// TIA Portal V19 export
FUNCTION "FC70_RecordData" : Void   // FC70, LAD
{ S7_Optimized_Access := 'TRUE' }
// stored: AutoNumber false, SetENOAutomatically false
   VAR_TEMP   // added for the SCL form of the ladder/FBD networks
      _w1 : Bool;
   END_VAR
BEGIN

REGION Network 1: Record Production data
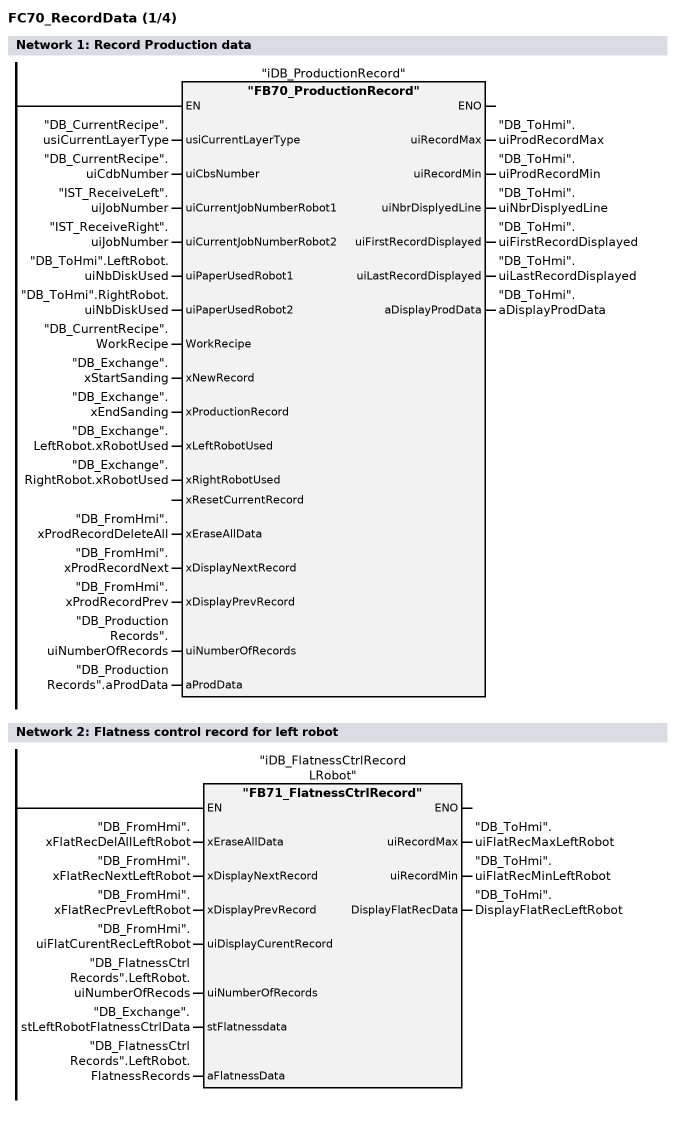
   RUNG wire#powerrail
      "iDB_ProductionRecord"(usiCurrentLayerType := "DB_CurrentRecipe".usiCurrentLayerType, uiCbsNumber := "DB_CurrentRecipe".uiCdbNumber, uiCurrentJobNumberRobot1 := "IST_ReceiveLeft".uiJobNumber, uiCurrentJobNumberRobot2 := "IST_ReceiveRight".uiJobNumber, uiPaperUsedRobot1 := "DB_ToHmi".LeftRobot.uiNbDiskUsed, uiPaperUsedRobot2 := "DB_ToHmi".RightRobot.uiNbDiskUsed, WorkRecipe := "DB_CurrentRecipe".WorkRecipe, xNewRecord := "DB_Exchange".xStartSanding, xProductionRecord := "DB_Exchange".xEndSanding, xLeftRobotUsed := "DB_Exchange".LeftRobot.xRobotUsed, xRightRobotUsed := "DB_Exchange".RightRobot.xRobotUsed, xResetCurrentRecord :=, xEraseAllData := "DB_FromHmi".xProdRecordDeleteAll, xDisplayNextRecord := "DB_FromHmi".xProdRecordNext, xDisplayPrevRecord := "DB_FromHmi".xProdRecordPrev, uiNumberOfRecords := "DB_ProductionRecords".uiNumberOfRecords, aProdData := "DB_ProductionRecords".aProdData, uiRecordMax => "DB_ToHmi".uiProdRecordMax, uiRecordMin => "DB_ToHmi".uiProdRecordMin, uiNbrDisplyedLine => "DB_ToHmi".uiNbrDisplyedLine, uiFirstRecordDisplayed => "DB_ToHmi".uiFirstRecordDisplayed, uiLastRecordDisplayed => "DB_ToHmi".uiLastRecordDisplayed, aDisplayProdData => "DB_ToHmi".aDisplayProdData)
   END_RUNG
   // the same network as SCL:
   "iDB_ProductionRecord"(usiCurrentLayerType := "DB_CurrentRecipe".usiCurrentLayerType,   // "FB70_ProductionRecord"
                          uiCbsNumber := "DB_CurrentRecipe".uiCdbNumber,
                          uiCurrentJobNumberRobot1 := "IST_ReceiveLeft".uiJobNumber,
                          uiCurrentJobNumberRobot2 := "IST_ReceiveRight".uiJobNumber,
                          uiPaperUsedRobot1 := "DB_ToHmi".LeftRobot.uiNbDiskUsed,
                          uiPaperUsedRobot2 := "DB_ToHmi".RightRobot.uiNbDiskUsed,
                          WorkRecipe := "DB_CurrentRecipe".WorkRecipe,
                          xNewRecord := "DB_Exchange".xStartSanding,
                          xProductionRecord := "DB_Exchange".xEndSanding,
                          xLeftRobotUsed := "DB_Exchange".LeftRobot.xRobotUsed,
                          xRightRobotUsed := "DB_Exchange".RightRobot.xRobotUsed,
                          xEraseAllData := "DB_FromHmi".xProdRecordDeleteAll,
                          xDisplayNextRecord := "DB_FromHmi".xProdRecordNext,
                          xDisplayPrevRecord := "DB_FromHmi".xProdRecordPrev,
                          uiNumberOfRecords := "DB_ProductionRecords".uiNumberOfRecords,
                          aProdData := "DB_ProductionRecords".aProdData,
                          uiRecordMax => "DB_ToHmi".uiProdRecordMax,
                          uiRecordMin => "DB_ToHmi".uiProdRecordMin,
                          uiNbrDisplyedLine => "DB_ToHmi".uiNbrDisplyedLine,
                          uiFirstRecordDisplayed => "DB_ToHmi".uiFirstRecordDisplayed,
                          uiLastRecordDisplayed => "DB_ToHmi".uiLastRecordDisplayed,
                          aDisplayProdData => "DB_ToHmi".aDisplayProdData);
END_REGION

REGION Network 2: Flatness control record for left robot
   RUNG wire#powerrail
      "iDB_FlatnessCtrlRecordLRobot"(xEraseAllData := "DB_FromHmi".xFlatRecDelAllLeftRobot, xDisplayNextRecord := "DB_FromHmi".xFlatRecNextLeftRobot, xDisplayPrevRecord := "DB_FromHmi".xFlatRecPrevLeftRobot, uiDisplayCurentRecord := "DB_FromHmi".uiFlatCurentRecLeftRobot, uiNumberOfRecords := "DB_FlatnessCtrlRecords".LeftRobot.uiNumberOfRecods, stFlatnessdata := "DB_Exchange".stLeftRobotFlatnessCtrlData, aFlatnessData := "DB_FlatnessCtrlRecords".LeftRobot.FlatnessRecords, uiRecordMax => "DB_ToHmi".uiFlatRecMaxLeftRobot, uiRecordMin => "DB_ToHmi".uiFlatRecMinLeftRobot, DisplayFlatRecData => "DB_ToHmi".DisplayFlatRecLeftRobot)
   END_RUNG
   // the same network as SCL:
   "iDB_FlatnessCtrlRecordLRobot"(xEraseAllData := "DB_FromHmi".xFlatRecDelAllLeftRobot,   // "FB71_FlatnessCtrlRecord"
                           xDisplayNextRecord := "DB_FromHmi".xFlatRecNextLeftRobot,
                           xDisplayPrevRecord := "DB_FromHmi".xFlatRecPrevLeftRobot,
                           uiDisplayCurentRecord := "DB_FromHmi".uiFlatCurentRecLeftRobot,
                           uiNumberOfRecords := "DB_FlatnessCtrlRecords".LeftRobot.uiNumberOfRecods,
                           stFlatnessdata := "DB_Exchange".stLeftRobotFlatnessCtrlData,
                           aFlatnessData := "DB_FlatnessCtrlRecords".LeftRobot.FlatnessRecords,
                           uiRecordMax => "DB_ToHmi".uiFlatRecMaxLeftRobot,
                           uiRecordMin => "DB_ToHmi".uiFlatRecMinLeftRobot,
                           DisplayFlatRecData => "DB_ToHmi".DisplayFlatRecLeftRobot);
END_REGION

REGION Network 3: Flatness control record for Right robot
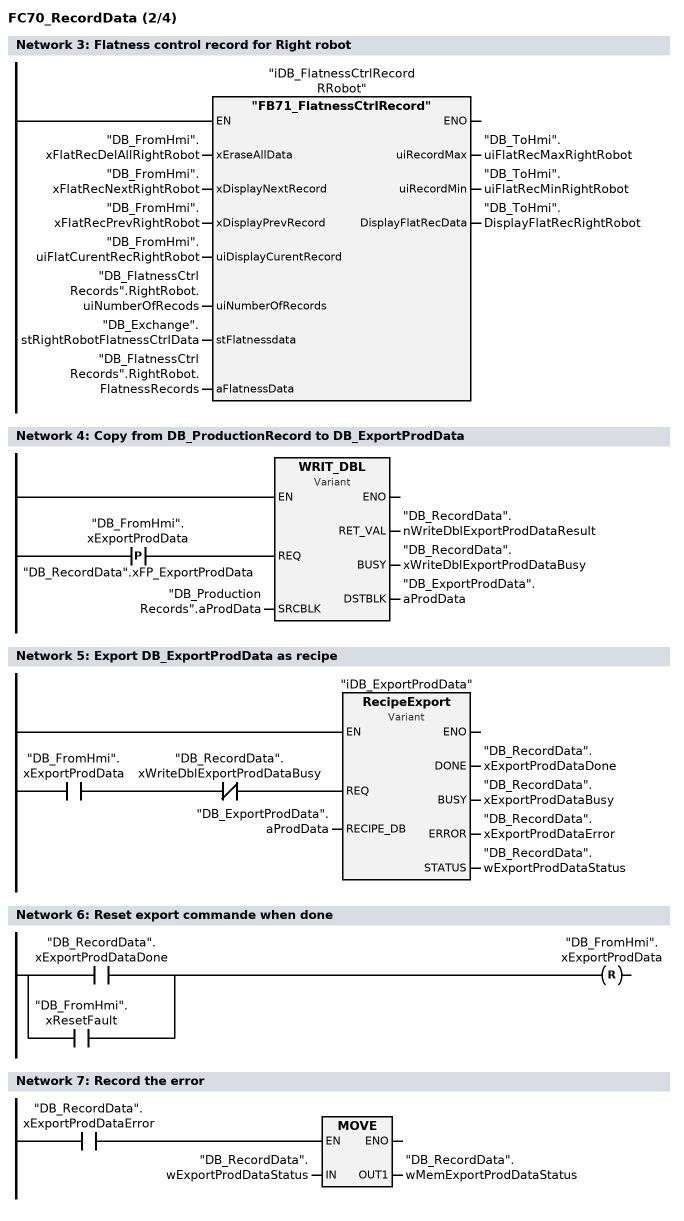
   RUNG wire#powerrail
      "iDB_FlatnessCtrlRecordRRobot"(xEraseAllData := "DB_FromHmi".xFlatRecDelAllRightRobot, xDisplayNextRecord := "DB_FromHmi".xFlatRecNextRightRobot, xDisplayPrevRecord := "DB_FromHmi".xFlatRecPrevRightRobot, uiDisplayCurentRecord := "DB_FromHmi".uiFlatCurentRecRightRobot, uiNumberOfRecords := "DB_FlatnessCtrlRecords".RightRobot.uiNumberOfRecods, stFlatnessdata := "DB_Exchange".stRightRobotFlatnessCtrlData, aFlatnessData := "DB_FlatnessCtrlRecords".RightRobot.FlatnessRecords, uiRecordMax => "DB_ToHmi".uiFlatRecMaxRightRobot, uiRecordMin => "DB_ToHmi".uiFlatRecMinRightRobot, DisplayFlatRecData => "DB_ToHmi".DisplayFlatRecRightRobot)
   END_RUNG
   // the same network as SCL:
   "iDB_FlatnessCtrlRecordRRobot"(xEraseAllData := "DB_FromHmi".xFlatRecDelAllRightRobot,   // "FB71_FlatnessCtrlRecord"
                           xDisplayNextRecord := "DB_FromHmi".xFlatRecNextRightRobot,
                           xDisplayPrevRecord := "DB_FromHmi".xFlatRecPrevRightRobot,
                           uiDisplayCurentRecord := "DB_FromHmi".uiFlatCurentRecRightRobot,
                           uiNumberOfRecords := "DB_FlatnessCtrlRecords".RightRobot.uiNumberOfRecods,
                           stFlatnessdata := "DB_Exchange".stRightRobotFlatnessCtrlData,
                           aFlatnessData := "DB_FlatnessCtrlRecords".RightRobot.FlatnessRecords,
                           uiRecordMax => "DB_ToHmi".uiFlatRecMaxRightRobot,
                           uiRecordMin => "DB_ToHmi".uiFlatRecMinRightRobot,
                           DisplayFlatRecData => "DB_ToHmi".DisplayFlatRecRightRobot);
END_REGION

REGION Network 4: Copy from DB_ProductionRecord to DB_ExportProdData
   RUNG wire#powerrail
      { S7_Templates := "[src_type := Variant, dest_type := Variant]" } WRIT_DBL(REQ := wire#w1, SRCBLK := "DB_ProductionRecords".aProdData, RET_VAL => "DB_RecordData".nWriteDblExportProdDataResult, BUSY => "DB_RecordData".xWriteDblExportProdDataBusy, DSTBLK => "DB_ExportProdData".aProdData)
   END_RUNG
   RUNG wire#powerrail
      P_Contact(operand := "DB_FromHmi".xExportProdData, bit := "DB_RecordData".xFP_ExportProdData)
   END_RUNG wire#w1
   // the same network as SCL:
   #_w1 := "DB_FromHmi".xExportProdData AND NOT "DB_RecordData".xFP_ExportProdData;   // rising edge of "DB_FromHmi".xExportProdData
   "DB_RecordData".xFP_ExportProdData := "DB_FromHmi".xExportProdData;
   "DB_RecordData".nWriteDblExportProdDataResult := WRIT_DBL(REQ := #_w1,
                           SRCBLK := "DB_ProductionRecords".aProdData,
                           BUSY => "DB_RecordData".xWriteDblExportProdDataBusy,
                           DSTBLK => "DB_ExportProdData".aProdData);
END_REGION

REGION Network 5: Export DB_ExportProdData as recipe
   RUNG wire#powerrail
      { S7_Templates := "recipe_type := Variant" } "iDB_ExportProdData".RecipeExport(REQ := wire#w1, RECIPE_DB := "DB_ExportProdData".aProdData, DONE => "DB_RecordData".xExportProdDataDone, BUSY => "DB_RecordData".xExportProdDataBusy, ERROR => "DB_RecordData".xExportProdDataError, STATUS => "DB_RecordData".wExportProdDataStatus)
   END_RUNG
   RUNG wire#powerrail
      Contact( "DB_FromHmi".xExportProdData )
      I_Contact( "DB_RecordData".xWriteDblExportProdDataBusy )
   END_RUNG wire#w1
   // the same network as SCL:
   "iDB_ExportProdData"(REQ := "DB_FromHmi".xExportProdData AND NOT "DB_RecordData".xWriteDblExportProdDataBusy,   // RecipeExport
                        RECIPE_DB := "DB_ExportProdData".aProdData,
                        DONE => "DB_RecordData".xExportProdDataDone,
                        BUSY => "DB_RecordData".xExportProdDataBusy,
                        ERROR => "DB_RecordData".xExportProdDataError,
                        STATUS => "DB_RecordData".wExportProdDataStatus);
END_REGION

REGION Network 6: Reset export commande when done
   RUNG wire#powerrail
      Contact( "DB_RecordData".xExportProdDataDone )
      wire#w1
      R_Coil( "DB_FromHmi".xExportProdData )
   END_RUNG
   RUNG wire#powerrail
      Contact( "DB_FromHmi".xResetFault )
   END_RUNG wire#w1
   // the same network as SCL:
   IF "DB_RecordData".xExportProdDataDone OR "DB_FromHmi".xResetFault THEN
       "DB_FromHmi".xExportProdData := FALSE;
   END_IF;
END_REGION

REGION Network 7: Record the error
   RUNG wire#powerrail
      Contact( "DB_RecordData".xExportProdDataError )
      Move(in := "DB_RecordData".wExportProdDataStatus, out1 => "DB_RecordData".wMemExportProdDataStatus)
   END_RUNG
   // the same network as SCL:
   IF "DB_RecordData".xExportProdDataError THEN
       "DB_RecordData".wMemExportProdDataStatus := "DB_RecordData".wExportProdDataStatus;
   END_IF;
END_REGION

REGION Network 8: Copy from DB_ProductionRecords to DB_ExportFlatCtrlRobot1
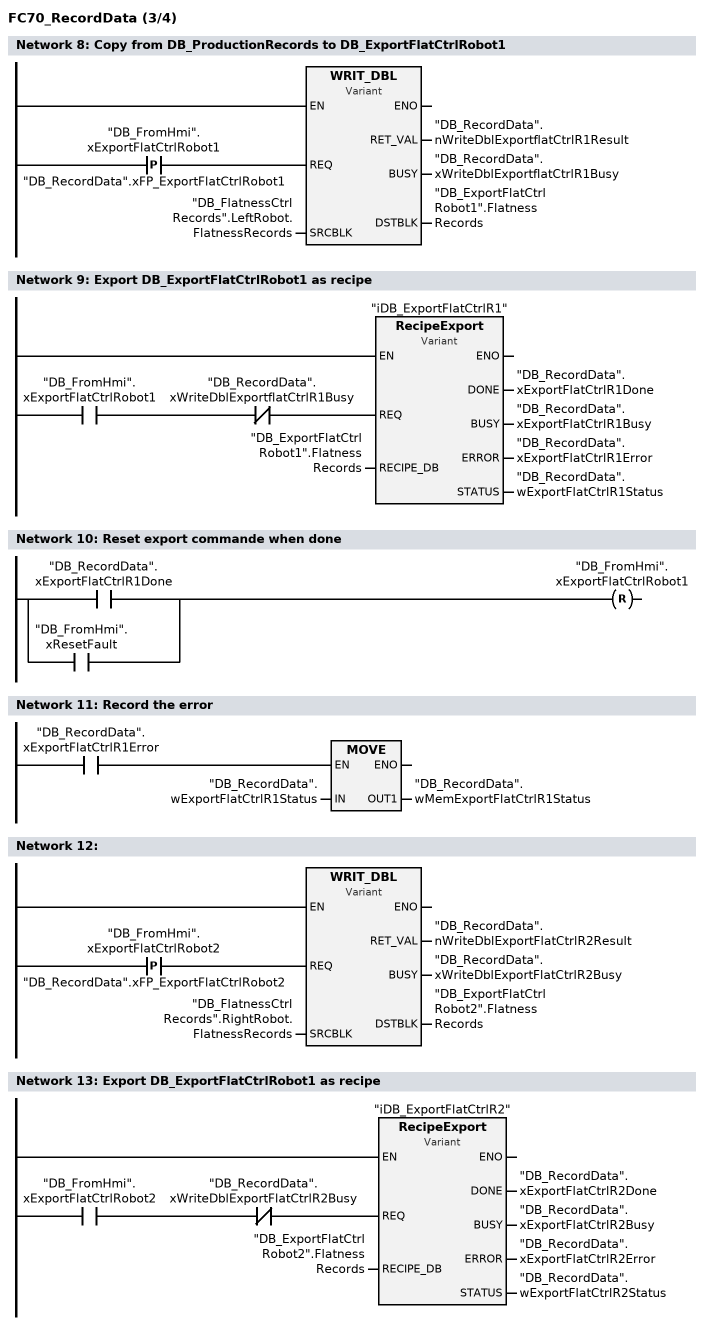
   RUNG wire#powerrail
      { S7_Templates := "[src_type := Variant, dest_type := Variant]" } WRIT_DBL(REQ := wire#w1, SRCBLK := "DB_FlatnessCtrlRecords".LeftRobot.FlatnessRecords, RET_VAL => "DB_RecordData".nWriteDblExportflatCtrlR1Result, BUSY => "DB_RecordData".xWriteDblExportflatCtrlR1Busy, DSTBLK => "DB_ExportFlatCtrlRobot1".FlatnessRecords)
   END_RUNG
   RUNG wire#powerrail
      P_Contact(operand := "DB_FromHmi".xExportFlatCtrlRobot1, bit := "DB_RecordData".xFP_ExportFlatCtrlRobot1)
   END_RUNG wire#w1
   // the same network as SCL:
   #_w1 := "DB_FromHmi".xExportFlatCtrlRobot1 AND NOT "DB_RecordData".xFP_ExportFlatCtrlRobot1;   // rising edge of "DB_FromHmi".xExportFlatCtrlRobot1
   "DB_RecordData".xFP_ExportFlatCtrlRobot1 := "DB_FromHmi".xExportFlatCtrlRobot1;
   "DB_RecordData".nWriteDblExportflatCtrlR1Result := WRIT_DBL(REQ := #_w1,
                           SRCBLK := "DB_FlatnessCtrlRecords".LeftRobot.FlatnessRecords,
                           BUSY => "DB_RecordData".xWriteDblExportflatCtrlR1Busy,
                           DSTBLK => "DB_ExportFlatCtrlRobot1".FlatnessRecords);
END_REGION

REGION Network 9: Export DB_ExportFlatCtrlRobot1 as recipe
   RUNG wire#powerrail
      { S7_Templates := "recipe_type := Variant" } "iDB_ExportFlatCtrlR1".RecipeExport(REQ := wire#w1, RECIPE_DB := "DB_ExportFlatCtrlRobot1".FlatnessRecords, DONE => "DB_RecordData".xExportFlatCtrlR1Done, BUSY => "DB_RecordData".xExportFlatCtrlR1Busy, ERROR => "DB_RecordData".xExportFlatCtrlR1Error, STATUS => "DB_RecordData".wExportFlatCtrlR1Status)
   END_RUNG
   RUNG wire#powerrail
      Contact( "DB_FromHmi".xExportFlatCtrlRobot1 )
      I_Contact( "DB_RecordData".xWriteDblExportflatCtrlR1Busy )
   END_RUNG wire#w1
   // the same network as SCL:
   "iDB_ExportFlatCtrlR1"(REQ := "DB_FromHmi".xExportFlatCtrlRobot1 AND NOT "DB_RecordData".xWriteDblExportflatCtrlR1Busy,   // RecipeExport
                          RECIPE_DB := "DB_ExportFlatCtrlRobot1".FlatnessRecords,
                          DONE => "DB_RecordData".xExportFlatCtrlR1Done,
                          BUSY => "DB_RecordData".xExportFlatCtrlR1Busy,
                          ERROR => "DB_RecordData".xExportFlatCtrlR1Error,
                          STATUS => "DB_RecordData".wExportFlatCtrlR1Status);
END_REGION

REGION Network 10: Reset export commande when done
   RUNG wire#powerrail
      Contact( "DB_RecordData".xExportFlatCtrlR1Done )
      wire#w1
      R_Coil( "DB_FromHmi".xExportFlatCtrlRobot1 )
   END_RUNG
   RUNG wire#powerrail
      Contact( "DB_FromHmi".xResetFault )
   END_RUNG wire#w1
   // the same network as SCL:
   IF "DB_RecordData".xExportFlatCtrlR1Done OR "DB_FromHmi".xResetFault THEN
       "DB_FromHmi".xExportFlatCtrlRobot1 := FALSE;
   END_IF;
END_REGION

REGION Network 11: Record the error
   RUNG wire#powerrail
      Contact( "DB_RecordData".xExportFlatCtrlR1Error )
      Move(in := "DB_RecordData".wExportFlatCtrlR1Status, out1 => "DB_RecordData".wMemExportFlatCtrlR1Status)
   END_RUNG
   // the same network as SCL:
   IF "DB_RecordData".xExportFlatCtrlR1Error THEN
       "DB_RecordData".wMemExportFlatCtrlR1Status := "DB_RecordData".wExportFlatCtrlR1Status;
   END_IF;
END_REGION

REGION Network 12
   RUNG wire#powerrail
      { S7_Templates := "[src_type := Variant, dest_type := Variant]" } WRIT_DBL(REQ := wire#w1, SRCBLK := "DB_FlatnessCtrlRecords".RightRobot.FlatnessRecords, RET_VAL => "DB_RecordData".nWriteDblExportFlatCtrlR2Result, BUSY => "DB_RecordData".xWriteDblExportFlatCtrlR2Busy, DSTBLK => "DB_ExportFlatCtrlRobot2".FlatnessRecords)
   END_RUNG
   RUNG wire#powerrail
      P_Contact(operand := "DB_FromHmi".xExportFlatCtrlRobot2, bit := "DB_RecordData".xFP_ExportFlatCtrlRobot2)
   END_RUNG wire#w1
   // the same network as SCL:
   #_w1 := "DB_FromHmi".xExportFlatCtrlRobot2 AND NOT "DB_RecordData".xFP_ExportFlatCtrlRobot2;   // rising edge of "DB_FromHmi".xExportFlatCtrlRobot2
   "DB_RecordData".xFP_ExportFlatCtrlRobot2 := "DB_FromHmi".xExportFlatCtrlRobot2;
   "DB_RecordData".nWriteDblExportFlatCtrlR2Result := WRIT_DBL(REQ := #_w1,
                           SRCBLK := "DB_FlatnessCtrlRecords".RightRobot.FlatnessRecords,
                           BUSY => "DB_RecordData".xWriteDblExportFlatCtrlR2Busy,
                           DSTBLK => "DB_ExportFlatCtrlRobot2".FlatnessRecords);
END_REGION

REGION Network 13: Export DB_ExportFlatCtrlRobot1 as recipe
   RUNG wire#powerrail
      { S7_Templates := "recipe_type := Variant" } "iDB_ExportFlatCtrlR2".RecipeExport(REQ := wire#w1, RECIPE_DB := "DB_ExportFlatCtrlRobot2".FlatnessRecords, DONE => "DB_RecordData".xExportFlatCtrlR2Done, BUSY => "DB_RecordData".xExportFlatCtrlR2Busy, ERROR => "DB_RecordData".xExportFlatCtrlR2Error, STATUS => "DB_RecordData".wExportFlatCtrlR2Status)
   END_RUNG
   RUNG wire#powerrail
      Contact( "DB_FromHmi".xExportFlatCtrlRobot2 )
      I_Contact( "DB_RecordData".xWriteDblExportFlatCtrlR2Busy )
   END_RUNG wire#w1
   // the same network as SCL:
   "iDB_ExportFlatCtrlR2"(REQ := "DB_FromHmi".xExportFlatCtrlRobot2 AND NOT "DB_RecordData".xWriteDblExportFlatCtrlR2Busy,   // RecipeExport
                          RECIPE_DB := "DB_ExportFlatCtrlRobot2".FlatnessRecords,
                          DONE => "DB_RecordData".xExportFlatCtrlR2Done,
                          BUSY => "DB_RecordData".xExportFlatCtrlR2Busy,
                          ERROR => "DB_RecordData".xExportFlatCtrlR2Error,
                          STATUS => "DB_RecordData".wExportFlatCtrlR2Status);
END_REGION

REGION Network 14: Reset export commande when done
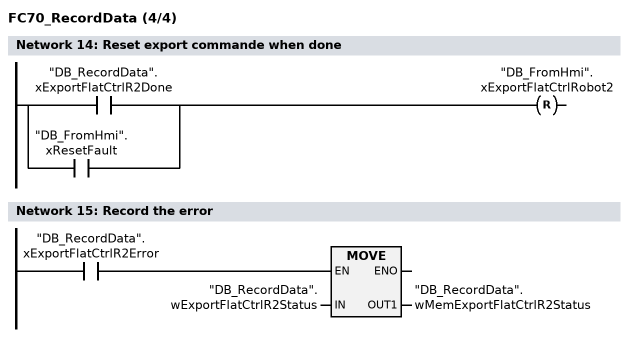
   RUNG wire#powerrail
      Contact( "DB_RecordData".xExportFlatCtrlR2Done )
      wire#w1
      R_Coil( "DB_FromHmi".xExportFlatCtrlRobot2 )
   END_RUNG
   RUNG wire#powerrail
      Contact( "DB_FromHmi".xResetFault )
   END_RUNG wire#w1
   // the same network as SCL:
   IF "DB_RecordData".xExportFlatCtrlR2Done OR "DB_FromHmi".xResetFault THEN
       "DB_FromHmi".xExportFlatCtrlRobot2 := FALSE;
   END_IF;
END_REGION

REGION Network 15: Record the error
   RUNG wire#powerrail
      Contact( "DB_RecordData".xExportFlatCtrlR2Error )
      Move(in := "DB_RecordData".wExportFlatCtrlR2Status, out1 => "DB_RecordData".wMemExportFlatCtrlR2Status)
   END_RUNG
   // the same network as SCL:
   IF "DB_RecordData".xExportFlatCtrlR2Error THEN
       "DB_RecordData".wMemExportFlatCtrlR2Status := "DB_RecordData".wExportFlatCtrlR2Status;
   END_IF;
END_REGION
END_FUNCTION
